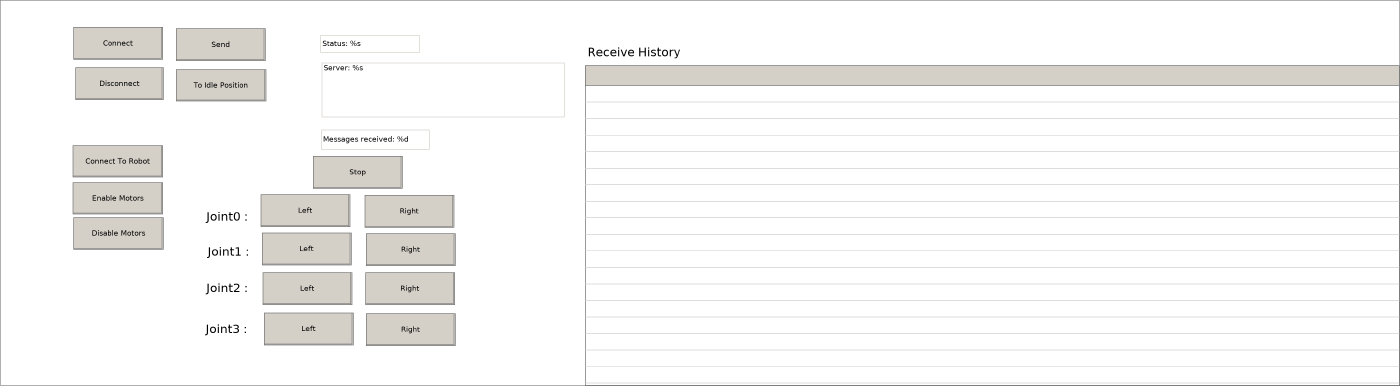
VISUALIZATION VisualizationControlPanel  // 2116x584
    Button (114,102 133x49), "Disconnect"
        tap MAIN.buttonDisconnectPressed
    Button (266,43 135x49), "Send"
        tap MAIN.buttonSendPressed
    Button (111,41 135x49), "Connect"
        tap MAIN.buttonConnectPressed
    Textfield (486,95 367x82), "Server: %s", text variable: MAIN.messageFromServer
    Textfield (485,196 164x30), "Messages received: %d", text variable: MAIN.totalMessagesFromServerCount
    Table (884,99 1232x485), data array: MAIN.messageHistoryArray
        p3854506369: MAIN.messageHistoryArray[INDEX].systemTimeString
        p1892666644: MAIN.messageHistoryArray[INDEX].message
        p511219082: Message
    Label (885,64 182x30), "Receive History"
    Button (110,220 136x48), "Connect To Robot"
        tap MAIN.buttonConnectToRobotPressed
    Button (266,105 136x48), "To Idle Position"
        tap MAIN.buttonDebugSendPressed
    Button (110,276 136x48), "Enable Motors"
        tap MAIN.buttonEnableMotorsPressed
    Textfield (484,53 150x26), "Status: %s", text variable: MAIN.connectionMessage
    Button (111,329 136x48), "Disable Motors"
        tap MAIN.buttonDisableMotorsPressed
    Button (394,294 135x49), "Left"
        tap MAIN.buttonLeft0Pressed
    Button (551,295 135x49), "Right"
        tap MAIN.buttonRight0Pressed
    Button (473,236 135x49), "Stop"
        tap MAIN.buttonStopPressed
    Label (311,366 90x30), "Joint1 :"
    Button (553,353 135x49), "Right"
        tap MAIN.buttonRight1Pressed
    Button (552,412 135x49), "Right"
        tap MAIN.buttonRight2Pressed
    Button (553,474 135x49), "Right"
        tap MAIN.buttonRight3Pressed
    Button (396,352 135x49), "Left"
        tap MAIN.buttonLeft1Pressed
    Button (397,412 135x49), "Left"
        tap MAIN.buttonLeft2Pressed
    Button (399,473 135x49), "Left"
        tap MAIN.buttonLeft3Pressed
    Label (309,313 90x30), "Joint0 :"
    Label (309,421 90x30), "Joint2 :"
    Label (308,483 90x30), "Joint3 :"
END_VISUALIZATION

(* stored: Version 1.1.0.1, ProductVersion 3.1.4024.12
   Visu VisualizationControlPanel: Id {65fbdb0c-c9af-43b6-9432-86e4c4c3ac9b} *)
